// Mitsubishi GX Works2 project: DZRN_DDRVA   PLC: FX3U/FX3UC

PROGRAM MAIN
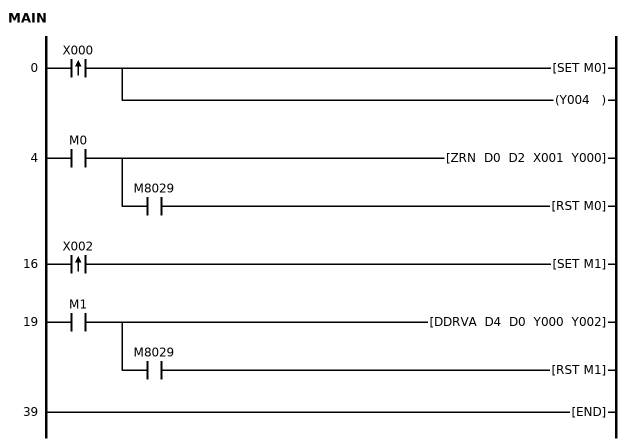
0     LDP     X000
      SET     M0
      OUT     Y004
4     LD      M0
      ZRN     D0 D2 X001 Y000
      AND     M8029
      RST     M0
16    LDP     X002
      SET     M1
19    LD      M1
      DDRVA   D4 D0 Y000 Y002
      AND     M8029
      RST     M1
39    END
END_PROGRAM
